(* IEC 61131-3 sources: repolevel_ST_code_completion/extract_code/轴控/FB105_轴控制集/FC12_设备手动, 4 files *)

(* ---- A03_气缸手动.st ---- *)
(**************************************************底膜部分*************************************************)
R_TRIG手动[1](CLK:= HMI_b取料气缸, Q=> );          F_TRIG手动[1](CLK:= HMI_b取料气缸, Q=> );
IF b非急停手动模式 AND R_TRIG手动[1].Q THEN
    DO_取料气缸:=TRUE;
END_IF
IF b非急停手动模式 AND F_TRIG手动[1].Q THEN
    DO_取料气缸:=FALSE;
END_IF

R_TRIG手动[2](CLK:= HMI_b纠偏气缸, Q=> );          F_TRIG手动[2](CLK:= HMI_b纠偏气缸, Q=> );
IF b非急停手动模式 AND R_TRIG手动[2].Q THEN
    DO_纠偏气缸:=TRUE;
END_IF
IF b非急停手动模式 AND F_TRIG手动[2].Q THEN
    DO_纠偏气缸:=FALSE;
END_IF

R_TRIG手动[3](CLK:= HMI_b挡料定位气缸, Q=> );      F_TRIG手动[3](CLK:= HMI_b挡料定位气缸, Q=> );
IF b非急停手动模式 AND R_TRIG手动[3].Q THEN
    DO_挡料定位气缸:=TRUE;
END_IF
IF b非急停手动模式 AND F_TRIG手动[3].Q THEN
    DO_挡料定位气缸:=FALSE;
END_IF

R_TRIG手动[4](CLK:= HMI_b翻板气缸, Q=> );          F_TRIG手动[4](CLK:= HMI_b翻板气缸, Q=> );
IF b非急停手动模式 AND R_TRIG手动[4].Q THEN
    DO_翻板气缸:=TRUE;
END_IF
IF b非急停手动模式 AND F_TRIG手动[4].Q THEN
    DO_翻板气缸:=FALSE;
END_IF

R_TRIG手动[5](CLK:= HMI_b侧压紧气缸, Q=> );         F_TRIG手动[5](CLK:= HMI_b侧压紧气缸, Q=> );
IF b非急停手动模式 AND R_TRIG手动[5].Q THEN
    DO_侧压紧气缸:=TRUE;
END_IF
IF b非急停手动模式 AND F_TRIG手动[5].Q THEN
    DO_侧压紧气缸:=FALSE;
END_IF

R_TRIG手动[6](CLK:= HMI_b左A包底气缸, Q=> );        F_TRIG手动[6](CLK:= HMI_b左A包底气缸, Q=> );
IF b非急停手动模式 AND R_TRIG手动[6].Q THEN
    DO_左A包底气缸:=TRUE;
END_IF
IF b非急停手动模式 AND F_TRIG手动[6].Q THEN
    DO_左A包底气缸:=FALSE;
END_IF

R_TRIG手动[7](CLK:= HMI_b右B包底气缸, Q=> );        F_TRIG手动[7](CLK:= HMI_b右B包底气缸, Q=> );
IF b非急停手动模式 AND R_TRIG手动[7].Q THEN
    DO_右B包底气缸:=TRUE;
END_IF
IF b非急停手动模式 AND F_TRIG手动[7].Q THEN
    DO_右B包底气缸:=FALSE;
END_IF

R_TRIG手动[8](CLK:= HMI_b上包底气缸, Q=> );         F_TRIG手动[8](CLK:= HMI_b上包底气缸, Q=> );
IF b非急停手动模式 AND R_TRIG手动[8].Q THEN
    DO_上包底气缸:=TRUE;
END_IF
IF b非急停手动模式 AND F_TRIG手动[8].Q THEN
    DO_上包底气缸:=FALSE;
END_IF

R_TRIG手动[9](CLK:= HMI_b下包底气缸, Q=> );         F_TRIG手动[9](CLK:= HMI_b下包底气缸, Q=> );
IF b非急停手动模式 AND R_TRIG手动[9].Q THEN
    DO_下包底气缸:=TRUE;
END_IF
IF b非急停手动模式 AND F_TRIG手动[9].Q THEN
    DO_下包底气缸:=FALSE;
END_IF

R_TRIG手动[10](CLK:= HMI_b出料推盒气缸, Q=> );      F_TRIG手动[10](CLK:= HMI_b出料推盒气缸, Q=> );
IF b非急停手动模式 AND R_TRIG手动[10].Q THEN
    DO_出料推盒气缸:=TRUE;
END_IF
IF b非急停手动模式 AND F_TRIG手动[10].Q THEN
    DO_出料推盒气缸:=FALSE;
END_IF

R_TRIG手动[11](CLK:= HMI_b包盒口升降气缸, Q=> );    F_TRIG手动[11](CLK:= HMI_b包盒口升降气缸, Q=> );
IF b非急停手动模式 AND R_TRIG手动[11].Q THEN
    DO_包盒口升降气缸:=TRUE;
END_IF
IF b非急停手动模式 AND F_TRIG手动[11].Q THEN
    DO_包盒口升降气缸:=FALSE;
END_IF

R_TRIG手动[12](CLK:= HMI_b包盒口下压气缸, Q=> );    F_TRIG手动[12](CLK:= HMI_b包盒口下压气缸, Q=> );
IF b非急停手动模式 AND R_TRIG手动[12].Q THEN
    DO_包盒口下压气缸:=TRUE;
END_IF
IF b非急停手动模式 AND F_TRIG手动[12].Q THEN
    DO_包盒口下压气缸:=FALSE;
END_IF

R_TRIG手动[13](CLK:= HMI_b翻底板气缸, Q=> );        F_TRIG手动[13](CLK:= HMI_b翻底板气缸, Q=> );
IF b非急停手动模式 AND R_TRIG手动[13].Q THEN
    DO_翻底板气缸:=TRUE;
END_IF
IF b非急停手动模式 AND F_TRIG手动[13].Q THEN
    DO_翻底板气缸:=FALSE;
END_IF

R_TRIG手动[14](CLK:= HMI_b推底板气缸, Q=> );        F_TRIG手动[14](CLK:= HMI_b推底板气缸, Q=> );
IF b非急停手动模式 AND R_TRIG手动[14].Q THEN
    DO_推底板气缸:=TRUE;
END_IF
IF b非急停手动模式 AND F_TRIG手动[14].Q THEN
    DO_推底板气缸:=FALSE;
END_IF

R_TRIG手动[15](CLK:= HMI_b模组吸底板气缸, Q=> );    F_TRIG手动[15](CLK:= HMI_b模组吸底板气缸, Q=> );
IF b非急停手动模式 AND R_TRIG手动[15].Q THEN
    DO_模组吸底板气缸:=TRUE;
END_IF
IF b非急停手动模式 AND F_TRIG手动[15].Q THEN
    DO_模组吸底板气缸:=FALSE;
END_IF

R_TRIG手动[16](CLK:= HMI_b包边纠偏上下气缸, Q=> );  F_TRIG手动[16](CLK:= HMI_b包边纠偏上下气缸, Q=> );
IF b非急停手动模式 AND R_TRIG手动[16].Q THEN
    DO_包边纠偏上下气缸:=TRUE;
END_IF
IF b非急停手动模式 AND F_TRIG手动[16].Q THEN
    DO_包边纠偏上下气缸:=FALSE;
END_IF

R_TRIG手动[17](CLK:= HMI_b包边纠偏左右气缸, Q=> );  F_TRIG手动[17](CLK:= HMI_b包边纠偏左右气缸, Q=> );
IF b非急停手动模式 AND R_TRIG手动[17].Q THEN
    DO_包边纠偏左右气缸:=TRUE;
END_IF
IF b非急停手动模式 AND F_TRIG手动[17].Q THEN
    DO_包边纠偏左右气缸:=FALSE;
END_IF

R_TRIG手动[18](CLK:= HMI_b包边压料气缸, Q=> );      F_TRIG手动[18](CLK:= HMI_b包边压料气缸, Q=> );
IF b非急停手动模式 AND R_TRIG手动[18].Q THEN
    DO_包边压料气缸:=TRUE;
END_IF
IF b非急停手动模式 AND F_TRIG手动[18].Q THEN
    DO_包边压料气缸:=FALSE;
END_IF

R_TRIG手动[19](CLK:= HMI_b折边上托气缸, Q=> );      F_TRIG手动[19](CLK:= HMI_b折边上托气缸, Q=> );
IF b非急停手动模式 AND R_TRIG手动[19].Q THEN
    DO_折边上托气缸:=TRUE;
END_IF
IF b非急停手动模式 AND F_TRIG手动[19].Q THEN
    DO_折边上托气缸:=FALSE;
END_IF

R_TRIG手动[20](CLK:= HMI_b包边铲边气缸, Q=> );      F_TRIG手动[20](CLK:= HMI_b包边铲边气缸, Q=> );
IF b非急停手动模式 AND R_TRIG手动[20].Q THEN
    DO_包边铲边气缸:=TRUE;
END_IF
IF b非急停手动模式 AND F_TRIG手动[20].Q THEN
    DO_包边铲边气缸:=FALSE;
END_IF

(* ---- A04_真空手动.st ---- *)
(**************************************************真空部分*************************************************)
R_TRIG手动[50](CLK:= HMI_b吸底板真空, Q=> );   F_TRIG手动[50](CLK:= HMI_b吸底板真空, Q=> );
IF b非急停手动模式 AND R_TRIG手动[50].Q THEN
    DO_吸底板真空:=TRUE;
END_IF
IF b非急停手动模式 AND F_TRIG手动[50].Q THEN
    DO_吸底板真空:=FALSE;
END_IF

R_TRIG手动[51](CLK:= HMI_b取面板真空, Q=> );   F_TRIG手动[51](CLK:= HMI_b取面板真空, Q=> );
IF b非急停手动模式 AND R_TRIG手动[51].Q THEN
    DO_取面板真空:=TRUE;
END_IF
IF b非急停手动模式 AND F_TRIG手动[51].Q THEN
    DO_取面板真空:=FALSE;
END_IF

R_TRIG手动[52](CLK:= HMI_bA模吸底板真空, Q=> );   F_TRIG手动[52](CLK:= HMI_bA模吸底板真空, Q=> );
IF b非急停手动模式 AND R_TRIG手动[52].Q THEN
    DO_A模吸底板真空:=TRUE;
END_IF
IF b非急停手动模式 AND F_TRIG手动[52].Q THEN
    DO_A模吸底板真空:=FALSE;
END_IF

R_TRIG手动[53](CLK:= HMI_bA模吸面板真空, Q=> );   F_TRIG手动[53](CLK:= HMI_bA模吸面板真空, Q=> );
IF b非急停手动模式 AND R_TRIG手动[53].Q THEN
    DO_A模吸面板真空:=TRUE;
END_IF
IF b非急停手动模式 AND F_TRIG手动[53].Q THEN
	DO_A模吸面板真空:=FALSE;
END_IF

R_TRIG手动[54](CLK:= HMI_bB模吸底板真空, Q=> );   F_TRIG手动[54](CLK:= HMI_bB模吸底板真空, Q=> );
IF b非急停手动模式 AND R_TRIG手动[54].Q THEN
    DO_B模吸底板真空:=TRUE;
END_IF
IF b非急停手动模式 AND F_TRIG手动[54].Q THEN
    DO_B模吸底板真空:=FALSE;
END_IF

R_TRIG手动[55](CLK:= HMI_bB模吸面板真空, Q=> );   F_TRIG手动[55](CLK:= HMI_bB模吸面板真空, Q=> );
IF b非急停手动模式 AND R_TRIG手动[55].Q THEN
    DO_B模吸面板真空:=TRUE;
END_IF
IF b非急停手动模式 AND F_TRIG手动[55].Q THEN
	DO_B模吸面板真空:=FALSE;
END_IF

(* ---- A05_其他手动.st ---- *)
(**************************************************其它部分*************************************************)
R_TRIG手动[80](CLK:= HMI_b真空泵, Q=> );        F_TRIG手动[80](CLK:= HMI_b真空泵, Q=> );
IF b非急停手动模式 AND R_TRIG手动[80].Q THEN
    DO_真空泵:=TRUE;
END_IF
IF b非急停手动模式 AND F_TRIG手动[80].Q THEN
    DO_真空泵:=FALSE;
END_IF

R_TRIG手动[81](CLK:= HMI_b出料皮带电机, Q=> );   F_TRIG手动[81](CLK:= HMI_b出料皮带电机, Q=> );
IF b非急停手动模式 AND R_TRIG手动[81].Q THEN
    DO_出料皮带电机:=TRUE;
END_IF
IF b非急停手动模式 AND F_TRIG手动[81].Q THEN
    DO_出料皮带电机:=FALSE;
END_IF

(* ---- FC12_设备手动.st ---- *)
PROGRAM FC12_设备手动
VAR
	R_TRIG手动: ARRAY[1..100] OF R_TRIG;
	F_TRIG手动: ARRAY[1..100] OF F_TRIG;
END_VAR

A01_气类操作();
A02_轴类手动();
A03_气缸手动();
A04_真空手动();
A05_其它手动();
